FUNCTION_BLOCK Fix1_FB
VAR_INPUT
CC1_Input 			: Fixture;					//Clamping Circuit-1
CC2_Input 			: Fixture;					//Clamping Circuit-2
CC3_Input 			: Fixture;					//Clamping Circuit-3
CC4_Input 			: Fixture;					//Clamping Circuit-4
CC5_Input 			: Fixture;					//Clamping Circuit-5
CC6_Input 			: Fixture;					//Clamping Circuit-6

Unit_Adv_Pb 		: BOOL;						//Fixture Cylinder Clamp Pb
Unit_Ret_Pb 		: BOOL;						//Fixture Cylinder Declamp Pb

Part1_Load_Comp 	: BOOL;						//OP710 Part-1 Load Complete
Part2_Load_Comp 	: BOOL;						//OP710 Part-2 Load Complete
Part1_Unload_Comp 	: BOOL;						//OP710 Part-1 Unload Complete
Part2_Unload_Comp 	: BOOL;						//OP710 Part-2 Unload Complete

Robot_Weld_Comp 	: BOOL;						//Robot Weld Complete
TR_0_Deg  			: BOOL;						//Trunnion at 0 degree
TR_20_Deg 			: BOOL;						//Trunnion at -20 degree
TR_45_Deg 			: BOOL;						//Trunnion at 45 degree
TR_80_Deg 			: BOOL;						//Trunnion at 80 degree

TT_180_Deg 		: BOOL;						//Trunnion at 180 degree
Roller_Down 		: BOOL;						//Roller Door Down position
Roller_Up 			: BOOL;						//Roller Door Up position
END_VAR

VAR_OUTPUT
CC1_Output 			: Fixture;							//Clamping Circuit-1
CC2_Output 			: Fixture;							//Clamping Circuit-2
CC3_Output 			: Fixture;							//Clamping Circuit-3
CC4_Output 			: Fixture;							//Clamping Circuit-4
CC5_Output 			: Fixture;							//Clamping Circuit-5
CC6_Output 			: Fixture;							//Clamping Circuit-6
Fix_Home_Position 	: BOOL;
Fix_Work_Position 	: BOOL;

END_VAR

VAR
Cyl_Delay 			: ARRAY [0..30] OF TON;
END_VAR

Fix_Home_Position := CC1_Output.Home_Position AND CC2_Output.Home_Position AND CC3_Output.Home_Position AND CC4_Output.Home_Position AND CC5_Output.Home_Position AND CC6_Output.Home_Position;
Fix_Work_Position := CC1_Output.Work_Position AND CC2_Output.Work_Position AND CC3_Output.Work_Position AND CC4_Output.Work_Position AND CC5_Output.Work_Position AND CC6_Output.Work_Position;

CASE Station_Mode OF
	
	0: 
	
	IF (CC1_Input.Manual_Sel AND Unit_Adv_Pb AND (NOT Unit_Ret_Pb) AND CC3_Output.Home_Position) THEN
		CC1_Output.o_Clamp_WP := TRUE;
		Cyl_Delay[0](IN:= CC1_Output.o_Clamp_WP, PT:= T#1S, Q=> , ET=> );
		IF Cyl_Delay[0].Q THEN
		CC1_Input.i_Clamp1_Fbk := CC1_Input.i_Clamp2_Fbk := CC1_Input.i_Clamp3_Fbk := CC1_Output.Work_Position := TRUE;
		CC1_Input.i_Declamp1_Fbk := CC1_Input.i_Declamp2_Fbk := CC1_Input.i_Declamp3_Fbk := CC1_Output.Home_Position := FALSE;
		CC1_Output.o_Clamp_WP := FALSE;
		END_IF
	ELSIF (CC1_Input.Manual_Sel AND Unit_Ret_Pb AND (NOT Unit_Adv_Pb) AND CC3_Output.Home_Position) THEN
		CC1_Output.o_Clamp_HP := TRUE;
		Cyl_Delay[1](IN:= CC1_Output.o_Clamp_HP, PT:= T#1S, Q=> , ET=> );
		IF Cyl_Delay[1].Q THEN
		CC1_Input.i_Declamp1_Fbk := CC1_Input.i_Declamp2_Fbk := CC1_Input.i_Declamp3_Fbk := CC1_Output.Home_Position := TRUE;
		CC1_Input.i_Clamp1_Fbk := CC1_Input.i_Clamp2_Fbk := CC1_Input.i_Clamp3_Fbk := CC1_Output.Work_Position := FALSE;
		CC1_Output.o_Clamp_HP := FALSE;
		END_IF
	END_IF
	
	IF (CC3_Input.Manual_Sel AND Unit_Adv_Pb AND (NOT Unit_Ret_Pb) AND CC1_Output.Work_Position) THEN
		CC3_Output.o_Clamp_WP := TRUE;
		Cyl_Delay[2](IN:= CC3_Output.o_Clamp_WP, PT:= T#1S, Q=> , ET=> );
		IF Cyl_Delay[2].Q THEN
		CC3_Input.i_Clamp1_Fbk := CC3_Input.i_Clamp2_Fbk := CC3_Input.i_Clamp3_Fbk := CC3_Output.Work_Position := TRUE;
		CC3_Input.i_Declamp1_Fbk := CC3_Input.i_Declamp2_Fbk := CC3_Input.i_Declamp3_Fbk := CC3_Output.Home_Position := FALSE;
		CC3_Output.o_Clamp_WP := FALSE;
		END_IF
	ELSIF (CC3_Input.Manual_Sel AND Unit_Ret_Pb AND (NOT Unit_Adv_Pb) AND CC1_Output.Work_Position) THEN
		CC3_Output.o_Clamp_HP := TRUE;
		Cyl_Delay[3](IN:= CC3_Output.o_Clamp_HP, PT:= T#1S, Q=> , ET=> );
		IF Cyl_Delay[3].Q THEN
		CC3_Input.i_Declamp1_Fbk := CC3_Input.i_Declamp2_Fbk := CC3_Input.i_Declamp3_Fbk := CC3_Output.Home_Position := TRUE;
		CC3_Input.i_Clamp1_Fbk := CC3_Input.i_Clamp2_Fbk := CC3_Input.i_Clamp3_Fbk := CC3_Output.Work_Position := FALSE;
		CC3_Output.o_Clamp_HP := FALSE;
		END_IF
	END_IF
	
	IF (CC5_Input.Manual_Sel AND Unit_Adv_Pb AND (NOT Unit_Ret_Pb) AND CC3_Output.Work_Position) THEN
		CC5_Output.o_Clamp_WP := TRUE;
		Cyl_Delay[4](IN:= CC5_Output.o_Clamp_WP, PT:= T#1S, Q=> , ET=> );
		IF Cyl_Delay[4].Q THEN
		CC5_Input.i_Clamp1_Fbk := CC5_Input.i_Clamp2_Fbk := CC5_Input.i_Clamp3_Fbk := CC5_Output.Work_Position := TRUE;
		CC5_Input.i_Declamp1_Fbk := CC5_Input.i_Declamp2_Fbk := CC5_Input.i_Declamp3_Fbk := CC5_Output.Home_Position := FALSE;
		CC5_Output.o_Clamp_WP := FALSE;
		END_IF
	ELSIF (CC5_Input.Manual_Sel AND Unit_Ret_Pb AND (NOT Unit_Adv_Pb) AND CC3_Output.Work_Position) THEN
		CC5_Output.o_Clamp_HP := TRUE;
		Cyl_Delay[5](IN:= CC5_Output.o_Clamp_HP, PT:= T#1S, Q=> , ET=> );
		IF Cyl_Delay[5].Q THEN
		CC5_Input.i_Declamp1_Fbk := CC5_Input.i_Declamp2_Fbk := CC5_Input.i_Declamp3_Fbk := CC5_Output.Home_Position := TRUE;
		CC5_Input.i_Clamp1_Fbk := CC5_Input.i_Clamp2_Fbk := CC5_Input.i_Clamp3_Fbk := CC5_Output.Work_Position := FALSE;
		CC5_Output.o_Clamp_HP := FALSE;
		END_IF
	END_IF
	
	IF (CC2_Input.Manual_Sel AND Unit_Adv_Pb AND (NOT Unit_Ret_Pb) AND CC5_Output.Work_Position) THEN
		CC2_Output.o_Clamp_WP := TRUE;
		Cyl_Delay[6](IN:= CC2_Output.o_Clamp_WP, PT:= T#1S, Q=> , ET=> );
		IF Cyl_Delay[6].Q THEN
		CC2_Input.i_Clamp1_Fbk := CC2_Input.i_Clamp2_Fbk := CC2_Input.i_Clamp3_Fbk := CC2_Output.Work_Position := TRUE;
		CC2_Input.i_Declamp1_Fbk := CC2_Input.i_Declamp2_Fbk := CC2_Input.i_Declamp3_Fbk := CC2_Output.Home_Position := FALSE;
		CC2_Output.o_Clamp_WP := FALSE;
		END_IF
	ELSIF (CC2_Input.Manual_Sel AND Unit_Ret_Pb AND (NOT Unit_Adv_Pb) AND CC5_Output.Work_Position) THEN
		CC2_Output.o_Clamp_HP := TRUE;
		Cyl_Delay[7](IN:= CC2_Output.o_Clamp_HP, PT:= T#1S, Q=> , ET=> );
		IF Cyl_Delay[7].Q THEN
		CC2_Input.i_Declamp1_Fbk := CC2_Input.i_Declamp2_Fbk := CC2_Input.i_Declamp3_Fbk := CC2_Output.Home_Position := TRUE;
		CC2_Input.i_Clamp1_Fbk := CC2_Input.i_Clamp2_Fbk := CC2_Input.i_Clamp3_Fbk := CC2_Output.Work_Position := FALSE;
		CC2_Output.o_Clamp_HP := FALSE;
		END_IF
	END_IF
	
	IF (CC4_Input.Manual_Sel AND Unit_Adv_Pb AND (NOT Unit_Ret_Pb) AND CC2_Output.Work_Position) THEN
		CC4_Output.o_Clamp_WP := TRUE;
		Cyl_Delay[8](IN:= CC4_Output.o_Clamp_WP, PT:= T#1S, Q=> , ET=> );
		IF Cyl_Delay[8].Q THEN
		CC4_Input.i_Clamp1_Fbk := CC4_Input.i_Clamp2_Fbk := CC4_Input.i_Clamp3_Fbk := CC4_Output.Work_Position := TRUE;
		CC4_Input.i_Declamp1_Fbk := CC4_Input.i_Declamp2_Fbk := CC4_Input.i_Declamp3_Fbk := CC4_Output.Home_Position := FALSE;
		CC4_Output.o_Clamp_WP := FALSE;
		END_IF
	ELSIF (CC4_Input.Manual_Sel AND Unit_Ret_Pb AND (NOT Unit_Adv_Pb) AND CC2_Output.Work_Position) THEN
		CC4_Output.o_Clamp_HP := TRUE;
		Cyl_Delay[9](IN:= CC4_Output.o_Clamp_HP, PT:= T#1S, Q=> , ET=> );
		IF Cyl_Delay[9].Q THEN
		CC4_Input.i_Declamp1_Fbk := CC4_Input.i_Declamp2_Fbk := CC4_Input.i_Declamp3_Fbk := CC4_Output.Home_Position := TRUE;
		CC4_Input.i_Clamp1_Fbk := CC4_Input.i_Clamp2_Fbk := CC4_Input.i_Clamp3_Fbk := CC4_Output.Work_Position := FALSE;
		CC4_Output.o_Clamp_HP := FALSE;
		END_IF
	END_IF
	
	IF (CC6_Input.Manual_Sel AND Unit_Adv_Pb AND (NOT Unit_Ret_Pb) AND CC4_Output.Work_Position) THEN
		CC6_Output.o_Clamp_WP := TRUE;
		Cyl_Delay[10](IN:= CC6_Output.o_Clamp_WP, PT:= T#1S, Q=> , ET=> );
		IF Cyl_Delay[10].Q THEN
		CC6_Input.i_Clamp1_Fbk := CC6_Input.i_Clamp2_Fbk := CC6_Input.i_Clamp3_Fbk := CC6_Output.Work_Position := TRUE;
		CC6_Input.i_Declamp1_Fbk := CC6_Input.i_Declamp2_Fbk := CC6_Input.i_Declamp3_Fbk := CC6_Output.Home_Position := FALSE;
		CC6_Output.o_Clamp_WP := FALSE;
		END_IF
	ELSIF (CC6_Input.Manual_Sel AND Unit_Ret_Pb AND (NOT Unit_Adv_Pb) AND CC4_Output.Work_Position) THEN
		CC6_Output.o_Clamp_HP := TRUE;
		Cyl_Delay[11](IN:= CC6_Output.o_Clamp_HP, PT:= T#1S, Q=> , ET=> );
		IF Cyl_Delay[11].Q THEN
		CC6_Input.i_Declamp1_Fbk := CC6_Input.i_Declamp2_Fbk := CC6_Input.i_Declamp3_Fbk := CC6_Output.Home_Position := TRUE;
		CC6_Input.i_Clamp1_Fbk := CC6_Input.i_Clamp2_Fbk := CC6_Input.i_Clamp3_Fbk := CC6_Output.Work_Position := FALSE;
		CC6_Output.o_Clamp_HP := FALSE;
		END_IF
	END_IF

	
	1:

	IF (Start_Pb AND CC1_Input.Auto_Sel AND TR_20_Deg AND Part1_Load_Comp AND CC3_Output.Home_Position) THEN
		CC1_Output.o_Clamp_WP := TRUE;
		Cyl_Delay[12](IN:= (CC1_Output.o_Clamp_WP), PT:= T#1S, Q=> , ET=> );
		IF Cyl_Delay[12].Q THEN
		CC1_Input.i_Declamp1_Fbk := CC1_Input.i_Declamp2_Fbk := CC1_Input.i_Declamp3_Fbk := CC1_Output.Home_Position := FALSE;
		CC1_Input.i_Clamp1_Fbk := CC1_Input.i_Clamp2_Fbk := CC1_Input.i_Clamp3_Fbk := CC1_Output.Work_Position := TRUE;
		CC1_Output.o_Clamp_WP := FALSE;
		END_IF
	END_IF
	IF (Start_Pb AND CC3_Input.Auto_Sel AND TR_20_Deg AND CC1_Output.Work_Position) THEN
		CC3_Output.o_Clamp_WP := TRUE;
		Cyl_Delay[13](IN:= CC3_Output.o_Clamp_WP, PT:= T#1S, Q=> , ET=> );
		IF Cyl_Delay[13].Q THEN
		CC3_Input.i_Declamp1_Fbk := CC3_Input.i_Declamp2_Fbk := CC3_Input.i_Declamp3_Fbk := CC3_Output.Home_Position := FALSE;
		CC3_Input.i_Clamp1_Fbk := CC3_Input.i_Clamp2_Fbk := CC3_Input.i_Clamp3_Fbk := CC3_Output.Work_Position := TRUE;
		CC3_Output.o_Clamp_WP := FALSE;
		END_IF
	END_IF
	IF (Start_Pb AND CC5_Input.Auto_Sel AND TR_20_Deg AND CC3_Output.Work_Position) THEN
		CC5_Output.o_Clamp_WP := TRUE;
		Cyl_Delay[14](IN:= CC5_Output.o_Clamp_WP, PT:= T#1S, Q=> , ET=> );
		IF Cyl_Delay[14].Q THEN
		CC5_Input.i_Declamp1_Fbk := CC5_Input.i_Declamp2_Fbk := CC5_Input.i_Declamp3_Fbk := CC5_Output.Home_Position := FALSE;
		CC5_Input.i_Clamp1_Fbk := CC5_Input.i_Clamp2_Fbk := CC5_Input.i_Clamp3_Fbk := CC5_Output.Work_Position := TRUE;
		CC5_Output.o_Clamp_WP := FALSE;
		END_IF
	END_IF
	IF (Start_Pb AND CC2_Input.Auto_Sel AND TR_80_Deg AND Part2_Load_Comp AND Roller_Down AND CC5_Output.Work_Position) THEN
		CC2_Output.o_Clamp_WP := TRUE;
		Cyl_Delay[15](IN:= CC2_Output.o_Clamp_WP, PT:= T#1S, Q=> , ET=> );
		IF Cyl_Delay[15].Q THEN
		CC2_Input.i_Declamp1_Fbk := CC2_Input.i_Declamp2_Fbk := CC2_Input.i_Declamp3_Fbk := CC2_Output.Home_Position := FALSE;
		CC2_Input.i_Clamp1_Fbk := CC2_Input.i_Clamp2_Fbk := CC2_Input.i_Clamp3_Fbk := CC2_Output.Work_Position := TRUE;
		CC2_Output.o_Clamp_WP := FALSE;
		END_IF
	END_IF
	IF (Start_Pb AND CC4_Input.Auto_Sel AND TR_80_Deg AND Roller_Down AND CC2_Output.Work_Position) THEN
		CC4_Output.o_Clamp_WP := TRUE;
		Cyl_Delay[16](IN:= CC4_Output.o_Clamp_WP, PT:= T#1S, Q=> , ET=> );
		IF Cyl_Delay[16].Q THEN
		CC4_Input.i_Declamp1_Fbk := CC4_Input.i_Declamp2_Fbk := CC4_Input.i_Declamp3_Fbk := CC4_Output.Home_Position := FALSE;
		CC4_Input.i_Clamp1_Fbk := CC4_Input.i_Clamp2_Fbk := CC4_Input.i_Clamp3_Fbk := CC4_Output.Work_Position := TRUE;
		CC4_Output.o_Clamp_WP := FALSE;
		END_IF
	END_IF
	IF (Start_Pb AND CC6_Input.Auto_Sel AND TR_80_Deg AND Roller_Down AND CC4_Output.Work_Position) THEN
		CC6_Output.o_Clamp_WP := TRUE;
		Cyl_Delay[17](IN:= CC6_Output.o_Clamp_WP, PT:= T#1S, Q=> , ET=> );
		IF Cyl_Delay[17].Q THEN
		CC6_Input.i_Declamp1_Fbk := CC6_Input.i_Declamp2_Fbk := CC6_Input.i_Declamp3_Fbk := CC6_Output.Home_Position := FALSE;
		CC6_Input.i_Clamp1_Fbk := CC6_Input.i_Clamp2_Fbk := CC6_Input.i_Clamp3_Fbk := CC6_Output.Work_Position := TRUE;
		CC6_Output.o_Clamp_WP := FALSE;
		END_IF
	END_IF
	IF (CC5_Input.Auto_Sel AND TT_180_Deg AND TR_0_Deg AND Robot_Weld_Comp) THEN
		CC5_Output.o_Clamp_HP := TRUE;
		Cyl_Delay[18](IN:= CC5_Output.o_Clamp_HP, PT:= T#1S, Q=> , ET=> );
		IF Cyl_Delay[18].Q THEN
		CC5_Input.i_Clamp1_Fbk := CC5_Input.i_Clamp2_Fbk := CC5_Input.i_Clamp3_Fbk := CC5_Output.Work_Position := FALSE;
		CC5_Input.i_Declamp1_Fbk := CC5_Input.i_Declamp2_Fbk := CC5_Input.i_Declamp3_Fbk := CC5_Output.Home_Position := TRUE;
		CC5_Output.o_clamp_HP := FALSE;
		END_IF
	END_IF
	IF (CC3_Input.Auto_Sel AND TT_180_Deg AND TR_0_Deg AND Robot_Weld_Comp) THEN
		CC3_Output.o_Clamp_HP := TRUE;
		Cyl_Delay[19](IN:= CC3_Output.o_Clamp_HP, PT:= T#1S, Q=> , ET=> );
		IF Cyl_Delay[19].Q THEN
		CC3_Input.i_Clamp1_Fbk := CC3_Input.i_Clamp2_Fbk := CC3_Input.i_Clamp3_Fbk := CC3_Output.Work_Position := FALSE;
		CC3_Input.i_Declamp1_Fbk := CC3_Input.i_Declamp2_Fbk := CC3_Input.i_Declamp3_Fbk := CC3_Output.Home_Position := TRUE;
		CC3_Output.o_clamp_HP := FALSE;
		END_IF
	END_IF
	IF (CC1_Input.Auto_Sel AND TT_180_Deg AND TR_0_Deg AND Robot_Weld_Comp) THEN
		CC1_Output.o_Clamp_HP := TRUE;
		Cyl_Delay[20](IN:= CC1_Output.o_Clamp_HP, PT:= T#1S, Q=> , ET=> );
		IF Cyl_Delay[20].Q THEN
		CC1_Input.i_Clamp1_Fbk := CC1_Input.i_Clamp2_Fbk := CC1_Input.i_Clamp3_Fbk := CC1_Output.Work_Position := FALSE;
		CC1_Input.i_Declamp1_Fbk := CC1_Input.i_Declamp2_Fbk := CC1_Input.i_Declamp3_Fbk := CC1_Output.Home_Position := TRUE;
		CC1_Output.o_clamp_HP := FALSE;
		END_IF
	END_IF
	IF (CC1_Output.Home_Position AND CC3_Output.Home_Position AND CC5_Output.Home_Position AND Roller_Up AND Part1_Unload_Comp AND TR_45_Deg AND TT_180_Deg AND Robot_Weld_Comp) THEN
		CC6_Output.o_Clamp_HP := TRUE;
		Cyl_Delay[21](IN:= CC6_Output.o_Clamp_HP, PT:= T#1S, Q=> , ET=> );
		IF Cyl_Delay[21].Q THEN
		CC6_Input.i_Clamp1_Fbk := CC6_Input.i_Clamp2_Fbk := CC6_Input.i_Clamp3_Fbk := CC6_Output.Work_Position := FALSE;
		CC6_Input.i_Declamp1_Fbk := CC6_Input.i_Declamp2_Fbk := CC6_Input.i_Declamp3_Fbk := CC6_Output.Home_Position := TRUE;
		CC6_Output.o_clamp_HP := FALSE;
		END_IF
	END_IF
	IF (CC6_Output.Home_Position AND Roller_Up AND Part1_Unload_Comp AND TR_45_Deg AND TT_180_Deg AND Robot_Weld_Comp) THEN
		CC4_Output.o_Clamp_HP := TRUE;
		Cyl_Delay[22](IN:= CC4_Output.o_Clamp_HP, PT:= T#1S, Q=> , ET=> );
		IF Cyl_Delay[22].Q THEN
		CC4_Input.i_Clamp1_Fbk := CC4_Input.i_Clamp2_Fbk := CC4_Input.i_Clamp3_Fbk := CC4_Output.Work_Position := FALSE;
		CC4_Input.i_Declamp1_Fbk := CC4_Input.i_Declamp2_Fbk := CC4_Input.i_Declamp3_Fbk := CC4_Output.Home_Position := TRUE;
		CC4_Output.o_clamp_HP := FALSE;
		END_IF
	END_IF
	IF (CC4_Output.Home_Position AND Roller_Up AND Part1_Unload_Comp AND TR_45_Deg AND TT_180_Deg AND Robot_Weld_Comp) THEN
		CC2_Output.o_Clamp_HP := TRUE;
		Cyl_Delay[23](IN:= CC2_Output.o_Clamp_HP, PT:= T#1S, Q=> , ET=> );
		IF Cyl_Delay[23].Q THEN
		CC2_Input.i_Clamp1_Fbk := CC2_Input.i_Clamp2_Fbk := CC2_Input.i_Clamp3_Fbk := CC2_Output.Work_Position := FALSE;
		CC2_Input.i_Declamp1_Fbk := CC2_Input.i_Declamp2_Fbk := CC2_Input.i_Declamp3_Fbk := CC2_Output.Home_Position := TRUE;
		CC2_Output.o_clamp_HP := FALSE;
		END_IF
	END_IF

END_CASE

END_FUNCTION_BLOCK

(* stored: Version 1.1.0.1, ProductVersion 3.1.4024.16
   POU Fix1_FB: Id {db3152cb-9a0e-4f53-85a7-c1cb9e2a4ac1}, SpecialFunc None *)
